// TIA Portal V19 export
TYPE "typeDataTransfer"
// stored: Access Published, Namespace Unit3
   STRUCT
      u3ToXyz : "Unit3.type_u3ToXyz";
      xyzToU3 { S7_SetPoint := 'True'} : "Unit3.type_XyzToU3";
   END_STRUCT;
END_TYPE
